TYPE RsiIncomingMsg :
STRUCT
END_STRUCT
END_TYPE

(* stored: Version 1.1.0.1, ProductVersion 3.1.4024.10
   DUT RsiIncomingMsg: Id {b5b7f54b-2aaa-454a-977c-e44c5d84ec64} *)
